// LS Electric XG5000 project: test2
// PLC NewPLC
// module base 0 slot 0: 입출력 모듈:XBC-DR20S (DC 24V 입력 12점, 릴레이 출력 8점)

PROGRAM NewProgram (task: 스캔 프로그램)

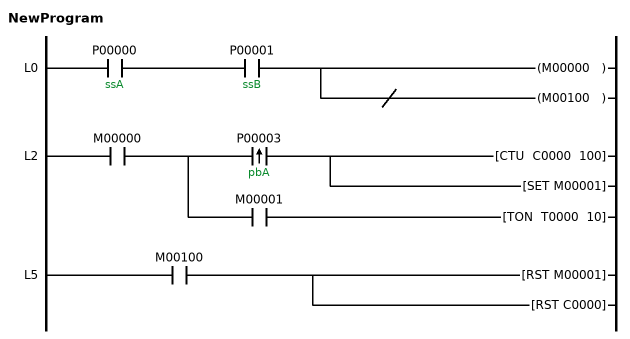
; L0
LOAD      P00000	// ssA
AND       P00001	// ssB
OUT       M00000
NOT
OUT       M00100
; L2
LOAD      M00000
MPUSH
ANDP      P00003	// pbA
CTU       C0000 100
SET       M00001
MPOP
AND       M00001
TON       T0000 10
; L5
LOAD      M00100
RST       M00001
RST       C0000

VARIABLES AND COMMENTS (devices not used above)
P00004	BIT	pbB
P00005	BIT	pbC
P00040	BIT	plA
P00041	BIT	plB
P00042	BIT	plC
P00043	BIT	plD
P00044	BIT	plE
P00002	BIT	ssC